{attribute addProperty BoxType "EPP9022-0060-0017"}
{attribute addProperty Id "Voltage_min_errorBIT10.1251Voltage_max_errorBIT10.1252Current_max_errorBIT10.1253Voltage_min_warningBIT10.1254Voltage_max_warningBIT10.1255Current_max_warningBIT10.1256Channel_errorBIT10.1257Channel_warningBIT10.1258TxPDO_StateBIT10.12515TxPDO_ToggleBIT10.12516"}
{attribute addProperty CRC "4045133654"}
{attribute addProperty SizeInBites "16"}
{attribute addProperty SizeInBytes "2"}
TYPE Status_F11BD756 :
STRUCT
	{attribute addProperty Name "Voltage_min_error"}
	Voltage_min_error : BIT;
	{attribute addProperty Name "Voltage_max_error"}
	Voltage_max_error : BIT;
	{attribute addProperty Name "Current_max_error"}
	Current_max_error : BIT;
	{attribute addProperty Name "Voltage_min_warning"}
	Voltage_min_warning : BIT;
	{attribute addProperty Name "Voltage_max_warning"}
	Voltage_max_warning : BIT;
	{attribute addProperty Name "Current_max_warning"}
	Current_max_warning : BIT;
	{attribute addProperty Name "Channel_error"}
	Channel_error : BIT;
	{attribute addProperty Name "Channel_warning"}
	Channel_warning : BIT;
	{attribute 'hide'}
	reserve_1_BIT_0 : BIT;
	{attribute 'hide'}
	reserve_1_BIT_1 : BIT;
	{attribute 'hide'}
	reserve_1_BIT_2 : BIT;
	{attribute 'hide'}
	reserve_1_BIT_3 : BIT;
	{attribute 'hide'}
	reserve_1_BIT_4 : BIT;
	{attribute 'hide'}
	reserve_1_BIT_5 : BIT;
	{attribute addProperty Name "TxPDO_State"}
	TxPDO_State : BIT;
	{attribute addProperty Name "TxPDO_Toggle"}
	TxPDO_Toggle : BIT;
END_STRUCT
END_TYPE

(* stored: Version 1.2.0.0, ProductVersion 3.1.4024.9
   DUT Status_F11BD756: Id {4203cafd-3fb7-4b78-82ba-74795615f9ef} *)
